// TIA Portal V20 export
DATA_BLOCK "BK23"   // DB142
// stored: MemoryReserve 100
   VAR
      "X10-1.SEPA CLAMP&CUTTER Z-AXIS LIMIT SENSOR(-)" : Bool := TRUE;
      "X11-1.SEPA CLAMP&CUTTER Z-AXIS LIMIT SENSOR(+)" : Bool := TRUE;
      "X12-1.SEPA CUTTER UP" : Bool := FALSE;
      "X13-1.SPARE" : Bool := FALSE;
      "X14-1.SPARE" : Bool := FALSE;
      "X15-1.SPARE" : Bool := FALSE;
      "X16-1.SEPA DETECT SENSOR" : Bool := FALSE;
      "X17-1.SPARE" : Bool := FALSE;
      "X10-2.CLAMP&CUTTER Z-AXIS HOME SENSOR" : Bool := TRUE;
      "X11-2.SPARE" : Bool := FALSE;
      "X12-2.SEPA CUTTER DOWN" : Bool := TRUE;
      "X13-2.SPARE" : Bool := FALSE;
      "X14-2.SPARE" : Bool := FALSE;
      "X15-2.SPARE" : Bool := FALSE;
      "X16-2.SPARE" : Bool := FALSE;
      "X17-2.SPARE" : Bool := FALSE;
   END_VAR
BEGIN
END_DATA_BLOCK
